/// default is port 851, every 10s.
FUNCTION_BLOCK T_WritePersistentData
VAR
	writePersistent: FB_WritePersistentData;
	writePeriod: TIME := TIME#10s0ms;
	adsPort: UINT := 851;
	writePersistTimer: TON;
END_VAR

// periodic force write of persistant variables.
writePersistTimer( IN := NOT writePersistTimer.Q, PT := writePeriod );
writePersistent( PORT:= adsPort, START := writePersistTimer.Q );

METHOD SetConfig : BOOL
VAR_INPUT
	/// How often to write data to persistent (default is 10S)/
	WritePeriod: TIME;
	/// which ads port (default is 851)
	AdsPort: UINT;
END_VAR
END_METHOD

END_FUNCTION_BLOCK

(* stored: Version 1.1.0.1, ProductVersion 3.1.4022.17
   POU T_WritePersistentData: Id {aa72b121-3a3c-4ff2-ba14-086414842741}, SpecialFunc None
   Method SetConfig: Id {e23e2b4c-1218-4ac3-a464-3a4fddad8077} *)
